FUNCTION_BLOCK TEST_ADP_SKT (* GUI for testing TEST_ADP as Socket *)
  (* Standard: 61499-1 *)
  (* Version 0.2, 2005-02-18, JHC, Rockwell Automation, Moved from "student" to "doc"; changed import from fb.rt.hmi to swing.. *)
  (* Version 0.1, 2003-08-17, JHC, Rockwell Automation, Moved from "book" to "student". *)
  (* Version 0.0, 2002-01-09, JHC, Rockwell Automation *)
  (* Compiler header: package fb.rt.doc; import fb.rt.swing.*; *)
  (* Compiler Java Sun JDK 1.4.2 *)
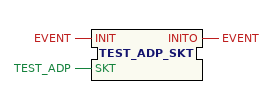
  EVENT_INPUT
    INIT : EVENT; (* Initialize GUI *)
  END_EVENT
  EVENT_OUTPUT
    INITO : EVENT; (* GUI Initialized *)
  END_EVENT
  SOCKETS
    SKT : TEST_ADP;
  END_SOCKETS
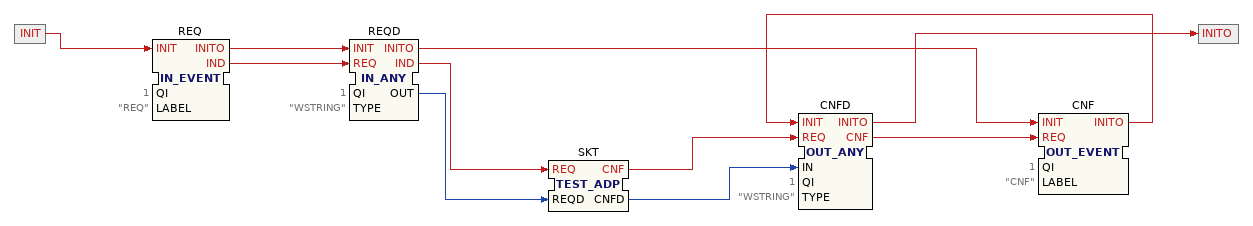
  FBS
    REQ : IN_EVENT(QI := 1, LABEL := "REQ");
    REQD : IN_ANY(QI := 1, TYPE := "WSTRING");
    CNF : OUT_EVENT(QI := 1, LABEL := "CNF");
    CNFD : OUT_ANY(QI := 1, TYPE := "WSTRING");
  END_FBS
  EVENT_CONNECTIONS
    INIT TO REQ.INIT;
    REQ.INITO TO REQD.INIT;
    REQD.INITO TO CNF.INIT;
    CNF.INITO TO CNFD.INIT;
    CNFD.INITO TO INITO;
    REQ.IND TO REQD.REQ;
    REQD.IND TO SKT.REQ;
    SKT.CNF TO CNFD.REQ;
    CNFD.CNF TO CNF.REQ;
  END_CONNECTIONS
  DATA_CONNECTIONS
    REQD.OUT TO SKT.REQD;
    SKT.CNFD TO CNFD.IN;
  END_CONNECTIONS
END_FUNCTION_BLOCK
